(* IEC 61131-3 sources: TIA2AX/tests/V18/test_projects/expected/HW_DiscoverGroups/PLC_3, 7 files *)

(* ---- HwIdentifiers.st ---- *)
TYPE
	HwIdentifiers : WORD
	(
		PLC_3_Rail_0 :=	WORD#256,
		PLC_3 :=	WORD#48,
		PLC_3_Card_reader_writer_1 :=	WORD#51,
		PLC_3_CPU_display_1 :=	WORD#54,
		PLC_3_PROFINET_interface_1 :=	WORD#64,
		PLC_3_PROFINET_interface_1_Port_1 :=	WORD#65,
		PLC_3_PROFINET_interface_1_Port_2 :=	WORD#66,
		PLC_3_10A_1 :=	WORD#257,
		PLC_3_10A_2 :=	WORD#258,
		PLC_3_10A_3 :=	WORD#259,
		PLC_3_10A_4 :=	WORD#260,
		PLC_3_10A_5 :=	WORD#261,
		PLC_3_10A_6 :=	WORD#262,
		PLC_3_10A_7 :=	WORD#263,
		PLC_3_10A_8 :=	WORD#264,
		PLC_3_10A_9 :=	WORD#265,
		PLC_3_10A_10 :=	WORD#266,
		PLC_3_10A_11 :=	WORD#267,
		PLC_3_10A_12 :=	WORD#268,
		_10A_17_Rack_0 :=	WORD#307,
		_10A_17 :=	WORD#308,
		_10A_17_10A_17 :=	WORD#309,
		_10A_17_PROFINET_interface :=	WORD#310,
		_10A_17_PROFINET_interface_Port_1 :=	WORD#311,
		_10A_17_PROFINET_interface_Port_2 :=	WORD#312,
		_10A_17_BA_2xRJ45 :=	WORD#311,
		_10A_17_10A_2 :=	WORD#313,
		_10A_17_10A_3 :=	WORD#314,
		_10A_17_10A_4 :=	WORD#315,
		_10A_17_10A_5 :=	WORD#316,
		_10A_17_10A_6 :=	WORD#317,
		_10A_17_10A_7 :=	WORD#318,
		_10A_17_10A_8 :=	WORD#319,
		_10A_17_10A_9 :=	WORD#320,
		_10A_17_10A_10 :=	WORD#321,
		_10A_17_10A_11 :=	WORD#322,
		_10A_17_Server_module_1 :=	WORD#323,
		_10A_21_Rack_0 :=	WORD#289,
		_10A_21 :=	WORD#290,
		_10A_21_10A_21 :=	WORD#291,
		_10A_21_PROFINET_interface :=	WORD#292,
		_10A_21_PROFINET_interface_Port_1 :=	WORD#293,
		_10A_21_PROFINET_interface_Port_2 :=	WORD#294,
		_10A_21_BA_2xRJ45 :=	WORD#293,
		_10A_21_10A_2 :=	WORD#295,
		_10A_21_10A_3 :=	WORD#296,
		_10A_21_10A_4 :=	WORD#297,
		_10A_21_10A_5 :=	WORD#298,
		_10A_21_10A_6 :=	WORD#299,
		_10A_21_10A_7 :=	WORD#300,
		_10A_21_10A_8 :=	WORD#301,
		_10A_21_10A_9 :=	WORD#302,
		_10A_21_10A_10 :=	WORD#303,
		_10A_21_10A_11 :=	WORD#304,
		_10A_21_Server_module_1 :=	WORD#305,
		_10A_13_Rack_0 :=	WORD#274,
		_10A_13 :=	WORD#275,
		_10A_13_10A_13 :=	WORD#276,
		_10A_13_PROFINET_interface :=	WORD#277,
		_10A_13_PROFINET_interface_Port_1 :=	WORD#278,
		_10A_13_PROFINET_interface_Port_2 :=	WORD#279,
		_10A_13_BA_2xRJ45 :=	WORD#278,
		_10A_13_10A_2 :=	WORD#280,
		_10A_13_10A_3 :=	WORD#281,
		_10A_13_10A_4 :=	WORD#282,
		_10A_13_10A_5 :=	WORD#283,
		_10A_13_10A_6 :=	WORD#284,
		_10A_13_10A_7 :=	WORD#285,
		_10A_13_10A_8 :=	WORD#286,
		_10A_13_10A_9 :=	WORD#287,
		_10A_13_10A_10 :=	WORD#270,
		_10A_13_10A_11 :=	WORD#271,
		_10A_13_Server_module_1 :=	WORD#272,
		NONE:= WORD#0
	);
END_TYPE

(* ---- HwInputs.st ---- *)
TYPE
	HwInputs : STRUCT
		PLC_3_10A_1 AT %B7 : WORD;
		PLC_3_10A_2 AT %B9 : WORD;
		PLC_3_10A_3 AT %B11 : WORD;
		PLC_3_10A_4 AT %B13 : WORD;
		PLC_3_10A_5 AT %B15 : WORD;
		PLC_3_10A_6 AT %B17 : WORD;
		_10A_17_10A_2 AT %B19 : BYTE;
		_10A_17_10A_3 AT %B20 : BYTE;
		_10A_17_10A_4 AT %B21 : BYTE;
		_10A_17_10A_5 AT %B22 : BYTE;
		_10A_17_10A_6 AT %B23 : BYTE;
		_10A_21_10A_2 AT %B24 : BYTE;
		_10A_21_10A_3 AT %B25 : BYTE;
		_10A_21_10A_4 AT %B26 : BYTE;
		_10A_21_10A_5 AT %B27 : BYTE;
		_10A_21_10A_6 AT %B28 : BYTE;
		_10A_13_10A_2 AT %B2 : BYTE;
		_10A_13_10A_3 AT %B3 : BYTE;
		_10A_13_10A_4 AT %B4 : BYTE;
		_10A_13_10A_5 AT %B5 : BYTE;
		_10A_13_10A_6 AT %B6 : BYTE;
	END_STRUCT;
END_TYPE

(* ---- HwOutputs.st ---- *)
TYPE
	HwOutputs : STRUCT
		PLC_3_10A_7 AT %B7 : WORD;
		PLC_3_10A_8 AT %B9 : WORD;
		PLC_3_10A_9 AT %B11 : WORD;
		PLC_3_10A_10 AT %B13 : WORD;
		PLC_3_10A_11 AT %B15 : WORD;
		PLC_3_10A_12 AT %B17 : WORD;
		_10A_17_10A_7 AT %B19 : BYTE;
		_10A_17_10A_8 AT %B20 : BYTE;
		_10A_17_10A_9 AT %B21 : BYTE;
		_10A_17_10A_10 AT %B22 : BYTE;
		_10A_17_10A_11 AT %B23 : BYTE;
		_10A_21_10A_7 AT %B24 : BYTE;
		_10A_21_10A_8 AT %B25 : BYTE;
		_10A_21_10A_9 AT %B26 : BYTE;
		_10A_21_10A_10 AT %B27 : BYTE;
		_10A_21_10A_11 AT %B28 : BYTE;
		_10A_13_10A_7 AT %B2 : BYTE;
		_10A_13_10A_8 AT %B3 : BYTE;
		_10A_13_10A_9 AT %B4 : BYTE;
		_10A_13_10A_10 AT %B5 : BYTE;
		_10A_13_10A_11 AT %B6 : BYTE;
	END_STRUCT;
END_TYPE

(* ---- PlcInputs.st ---- *)
TYPE
	PlcInputs : STRUCT
		PLC_3_10A_1 : WORD;
		PLC_3_10A_2 : WORD;
		PLC_3_10A_3 : WORD;
		PLC_3_10A_4 : WORD;
		PLC_3_10A_5 : WORD;
		PLC_3_10A_6 : WORD;
		_10A_17_10A_2 : BYTE;
		_10A_17_10A_3 : BYTE;
		_10A_17_10A_4 : BYTE;
		_10A_17_10A_5 : BYTE;
		_10A_17_10A_6 : BYTE;
		_10A_21_10A_2 : BYTE;
		_10A_21_10A_3 : BYTE;
		_10A_21_10A_4 : BYTE;
		_10A_21_10A_5 : BYTE;
		_10A_21_10A_6 : BYTE;
		_10A_13_10A_2 : BYTE;
		_10A_13_10A_3 : BYTE;
		_10A_13_10A_4 : BYTE;
		_10A_13_10A_5 : BYTE;
		_10A_13_10A_6 : BYTE;
	END_STRUCT;
END_TYPE

(* ---- PlcOutputs.st ---- *)
TYPE
	PlcOutputs : STRUCT
		PLC_3_10A_7 : WORD;
		PLC_3_10A_8 : WORD;
		PLC_3_10A_9 : WORD;
		PLC_3_10A_10 : WORD;
		PLC_3_10A_11 : WORD;
		PLC_3_10A_12 : WORD;
		_10A_17_10A_7 : BYTE;
		_10A_17_10A_8 : BYTE;
		_10A_17_10A_9 : BYTE;
		_10A_17_10A_10 : BYTE;
		_10A_17_10A_11 : BYTE;
		_10A_21_10A_7 : BYTE;
		_10A_21_10A_8 : BYTE;
		_10A_21_10A_9 : BYTE;
		_10A_21_10A_10 : BYTE;
		_10A_21_10A_11 : BYTE;
		_10A_13_10A_7 : BYTE;
		_10A_13_10A_8 : BYTE;
		_10A_13_10A_9 : BYTE;
		_10A_13_10A_10 : BYTE;
		_10A_13_10A_11 : BYTE;
	END_STRUCT;
END_TYPE

(* ---- CopyInputs.st ---- *)
FUNCTION CopyInputs
	VAR_EXTERNAL
		HwInputs : HwInputs;
		PlcInputs : PlcInputs;
	END_VAR
	PlcInputs.PLC_3_10A_1 := HwInputs.PLC_3_10A_1;
	PlcInputs.PLC_3_10A_2 := HwInputs.PLC_3_10A_2;
	PlcInputs.PLC_3_10A_3 := HwInputs.PLC_3_10A_3;
	PlcInputs.PLC_3_10A_4 := HwInputs.PLC_3_10A_4;
	PlcInputs.PLC_3_10A_5 := HwInputs.PLC_3_10A_5;
	PlcInputs.PLC_3_10A_6 := HwInputs.PLC_3_10A_6;
	PlcInputs._10A_17_10A_2 := HwInputs._10A_17_10A_2;
	PlcInputs._10A_17_10A_3 := HwInputs._10A_17_10A_3;
	PlcInputs._10A_17_10A_4 := HwInputs._10A_17_10A_4;
	PlcInputs._10A_17_10A_5 := HwInputs._10A_17_10A_5;
	PlcInputs._10A_17_10A_6 := HwInputs._10A_17_10A_6;
	PlcInputs._10A_21_10A_2 := HwInputs._10A_21_10A_2;
	PlcInputs._10A_21_10A_3 := HwInputs._10A_21_10A_3;
	PlcInputs._10A_21_10A_4 := HwInputs._10A_21_10A_4;
	PlcInputs._10A_21_10A_5 := HwInputs._10A_21_10A_5;
	PlcInputs._10A_21_10A_6 := HwInputs._10A_21_10A_6;
	PlcInputs._10A_13_10A_2 := HwInputs._10A_13_10A_2;
	PlcInputs._10A_13_10A_3 := HwInputs._10A_13_10A_3;
	PlcInputs._10A_13_10A_4 := HwInputs._10A_13_10A_4;
	PlcInputs._10A_13_10A_5 := HwInputs._10A_13_10A_5;
	PlcInputs._10A_13_10A_6 := HwInputs._10A_13_10A_6;
END_FUNCTION

(* ---- CopyOutputs.st ---- *)
FUNCTION CopyOutputs
	VAR_EXTERNAL
		HwOutputs : HwOutputs;
		PlcOutputs : PlcOutputs;
	END_VAR
	HwOutputs.PLC_3_10A_7 := PlcOutputs.PLC_3_10A_7;
	HwOutputs.PLC_3_10A_8 := PlcOutputs.PLC_3_10A_8;
	HwOutputs.PLC_3_10A_9 := PlcOutputs.PLC_3_10A_9;
	HwOutputs.PLC_3_10A_10 := PlcOutputs.PLC_3_10A_10;
	HwOutputs.PLC_3_10A_11 := PlcOutputs.PLC_3_10A_11;
	HwOutputs.PLC_3_10A_12 := PlcOutputs.PLC_3_10A_12;
	HwOutputs._10A_17_10A_7 := PlcOutputs._10A_17_10A_7;
	HwOutputs._10A_17_10A_8 := PlcOutputs._10A_17_10A_8;
	HwOutputs._10A_17_10A_9 := PlcOutputs._10A_17_10A_9;
	HwOutputs._10A_17_10A_10 := PlcOutputs._10A_17_10A_10;
	HwOutputs._10A_17_10A_11 := PlcOutputs._10A_17_10A_11;
	HwOutputs._10A_21_10A_7 := PlcOutputs._10A_21_10A_7;
	HwOutputs._10A_21_10A_8 := PlcOutputs._10A_21_10A_8;
	HwOutputs._10A_21_10A_9 := PlcOutputs._10A_21_10A_9;
	HwOutputs._10A_21_10A_10 := PlcOutputs._10A_21_10A_10;
	HwOutputs._10A_21_10A_11 := PlcOutputs._10A_21_10A_11;
	HwOutputs._10A_13_10A_7 := PlcOutputs._10A_13_10A_7;
	HwOutputs._10A_13_10A_8 := PlcOutputs._10A_13_10A_8;
	HwOutputs._10A_13_10A_9 := PlcOutputs._10A_13_10A_9;
	HwOutputs._10A_13_10A_10 := PlcOutputs._10A_13_10A_10;
	HwOutputs._10A_13_10A_11 := PlcOutputs._10A_13_10A_11;
END_FUNCTION
